TYPE ST_CODetectors :
STRUCT
	State 			: 	eCOAlarmStatus;
	b_CoValuesOK	: 	BOOL;
	Value 			:  	ARRAY[0..2] OF REAL;	//-1 if inoperative.
END_STRUCT
END_TYPE

(* stored: Version 1.1.0.1, ProductVersion 3.1.4024.12
   DUT ST_CODetectors: Id {4e68ee4d-cee5-48ad-9611-61222ca54397} *)
